// TwinCAT 3 PLC project Test_Proj
// ProgramVersion: 3.1.4026.25
// libraries:
//   Base Library, * (Beckhoff UK)
//   Eventlogger Library, * (Beckhoff UK)
//   Tc2_MC2, * (Beckhoff Automation GmbH)
//   Tc2_Standard, * (Beckhoff Automation GmbH)
//   Tc2_System, * (Beckhoff Automation GmbH)
//   Tc3_PlcTestSuite, * (Simmel)
//   [Motion Library], * (Beckhoff UK)
// project tree:
//   Manual Testing/ IntegrationTestSuite.TcPOU
//   / PlcTask.TcTTO
//   POUs/ MAIN.TcPOU
//   TestSuites/ AxisAbsTestSuite.TcPOU, AxisHaltTestSuite.TcPOU, AxisJogTestSuite.TcPOU, AxisModTestSuite.TcPOU, AxisPowerTestSuite.TcPOU, AxisRelTestSuite.TcPOU, AxisResetTestSuite.TcPOU, AxisTestSuite.TcPOU, GearOperationTestSuite.TcPOU, AxisVelocityTestSuite.TcPOU, SoEResetTestSuite.TcPOU
//   Stubs/ StubTask.TcPOU
// real-time tasks:
//   TASK PlcTask: cycle T#10ms, priority 20, ADS port 350
// motion (NC):
//   TASK NC-Task 1 SAF: cycle T#2ms, priority 4, ADS port 501
//   TASK NC-Task 1 SVB: cycle T#10ms, priority 8, ADS port 511
//   AXIS Axis 1 (id 1)
//     General: UnitName=°
//     Dynamic: Acceleration=90000, Deceleration=90000, Jerk=270000
//     Velo: RefSearch=600, RefSync=600, SlowManual=3000, FastManual=18000, Fast=60000, Maximum=60000
//     OtherSettings: AllowMotionCmdToSlave=true
//     encoder EncType=19
//       EncPara: ScaleFactorNumerator=360, ScaleFactorDenominator=1048576, MaxCount=#xffffffff
//     drive DrvType=16
//       DrvPara: MaxCount=#xffffffff, DriveControlDWord=#x00020100
//         Analog: VeloReferenz=66000, VeloScale=32, TorqueSetpointScale=10, ScaleFactorActTorque=0.1
//         TimeComp: TaskDelayCycles=1
//     controller CtrType=1
//       CtrPara: PriorControlFactor=1
//         Observer: BandWidth=20
//   AXIS Axis 2 (id 2)
//     OtherSettings: AllowMotionCmdToSlave=true
//     encoder EncType=1
//     drive DrvType=5
//       Analog: TorqueSetpointScale=10, ScaleFactorActTorque=0.1
//     controller CtrType=1
//       CtrPara: PriorControlFactor=1
//         Observer: BandWidth=20
// I/O:
//   DEVICE Device 2 (EtherCAT), AmsNetId 10.201.62.134.3.1
//     Term 1 (EK1100) [EK1100 EtherCAT Coupler (2A E-Bus)]
//       Term 2 (EL9227-5500) [EL9227-5500 Overcurrent protection 24V DC, 2Ch., max. 10A (sum), adjustable, extended functionalities]
//       Term 3 (EL1004) [EL1004 4Ch. Dig. Input 24V, 3ms]
//       Term 4 (EL2004) [EL2004 4Ch. Dig. Output 24V, 0.5A]
//       Term 5 (EL7211-0010) [EL7211-0010 1Ch. MDP742 Servo motor output stage with OCT (50V, 4.5A RMS)]
//       Term 6 (EL9011) [EL9011 End Terminal]
// variable links:
//   (this object) <-> Device 2 (EtherCAT)/Term 1 (EK1100)/Term 5 (EL7211-0010)
//     Drive/Inputs/In/nDataIn1 <-> DRV Following error actual value/Following error actual value
//     Drive/Inputs/In/nDcOutputTime <-> InfoData/DcOutputShift
//     Drive/Inputs/In/nState1 <-> DRV Statusword/Statusword
//     Drive/Inputs/In/nState2 <-> DRV Statusword/Statusword @bit 8
//     Drive/Inputs/In/nState4 @bit 1 <-> WcState/InputToggle
//     Drive/Inputs/In/nState4 <-> WcState/WcState
//     Drive/Outputs/Out/nCtrl1 <-> DRV Controlword/Controlword
//     Drive/Outputs/Out/nCtrl2 <-> DRV Controlword/Controlword @bit 8
//     Drive/Outputs/Out/nDataOut1 <-> DRV Target position/Target position
//     Enc/Inputs/In/nDataIn1 <-> FB Position/Position
//     Enc/Inputs/In/nDcInputTime <-> InfoData/DcInputShift
//     Enc/Inputs/In/nState4 @bit 1 <-> WcState/InputToggle
//     Enc/Inputs/In/nState4 <-> WcState/WcState
//   Test_Proj Instance <-> NC-Task 1 SAF/Axes/Axis 1
//     PlcTask Inputs/MAIN.Integration_TestSuite.StubAxis.NcToPlc <-> Outputs/ToPlc
//     PlcTask Outputs/MAIN.Integration_TestSuite.StubAxis.PlcToNc <-> Inputs/FromPlc
//   Test_Proj Instance <-> NC-Task 1 SAF/Axes/Axis 2
//     PlcTask Inputs/MAIN.Integration_TestSuite.gearSlave.NcToPlc <-> Outputs/ToPlc
//     PlcTask Outputs/MAIN.Integration_TestSuite.gearSlave.PlcToNc <-> Inputs/FromPlc
//   Test_Proj Instance <-> Test_Proj/Test_Proj Instance
//     PlcTask Inputs/MAIN.GearOperation_TestSuite.StubAxisRef1.NcToPlc/CoupleState <-> PlcTask Outputs/MAIN.GearOperation_TestSuite.GearAxisCoupledFeedback
//     PlcTask Inputs/MAIN.GearOperation_TestSuite.StubAxisRef1.NcToPlc/StateDWord <-> PlcTask Outputs/MAIN.GearOperation_TestSuite.GearAxisMotionFeedback
//     PlcTask Inputs/MAIN.Halt_TestSuite.StubAxis.NcToPlc/StateDWord <-> PlcTask Outputs/MAIN.Halt_TestSuite.HaltAxisStatusFeedback
//     PlcTask Outputs/MAIN.GearOperation_TestSuite.GearAxisCoupledFeedback <-> PlcTask Inputs/MAIN.GearOperation_TestSuite.StubAxisRef1.NcToPlc/CoupleState
//     PlcTask Outputs/MAIN.GearOperation_TestSuite.GearAxisMotionFeedback <-> PlcTask Inputs/MAIN.GearOperation_TestSuite.StubAxisRef1.NcToPlc/StateDWord
//     PlcTask Outputs/MAIN.Halt_TestSuite.HaltAxisStatusFeedback <-> PlcTask Inputs/MAIN.Halt_TestSuite.StubAxis.NcToPlc/StateDWord

CONFIGURATION Test_Proj
    RESOURCE PLC ON TwinCAT3
        TASK PlcTask(INTERVAL := T#10ms, PRIORITY := 20);
        PROGRAM MAIN WITH PlcTask : MAIN;
    END_RESOURCE
END_CONFIGURATION

// ---- POUs/MAIN.TcPOU
PROGRAM MAIN
VAR
	Power_TestSuite : AxisPowerTestSuite;
	Reset_TestSuite : AxisResetTestSuite;
	Halt_TestSuite : AxisHaltTestSuite;
	Axis_TestSuite : AxisTestSuite;
	AxisJog_TestSuite : AxisJogTestSuite;
	AxisVelo_TestSuite : AxisVelocityTestSuite;
	AxisAbs_TestSuite : AxisAbsTestSuite;
	AxisMod_TestSuite : AxisModTestSuite;
	AxisRel_TestSuite : AxisRelTestSuite;
	GearOperation_TestSuite : GearOperationTestSuite;
	SoEReset_TestSuite : SoEResetTestSuite;
	ReRun: BOOL;
	i : INT;
	Integration_TestSuite : IntegrationTestSuite;
END_VAR

Power_TestSuite();
Reset_TestSuite();
Halt_TestSuite();
Axis_TestSuite();
AxisJog_TestSuite();
AxisVelo_TestSuite();
AxisAbs_TestSuite();
AxisMod_TestSuite();
AxisRel_TestSuite();
GearOperation_TestSuite();
SoEReset_TestSuite();

Integration_TestSuite();

END_PROGRAM

// ---- TestSuites/AxisPowerTestSuite.TcPOU
FUNCTION_BLOCK AxisPowerTestSuite
VAR
	StubAxis : AXIS_REF;
	iStubTask : I_Task;
	TestAxisPower : EnableDisableTask := (AxisRef := StubAxis);
	ObjTestSuite : TestSuite<TestSuiteParameter.MaxTestCount>(ResultFile := JUnitResultFile) := (TestSuiteName := 'Object Test Suite');
END_VAR

DoesAxisAcceptEnable_Test();
RejectDisableWhenDisabled_Test();
RejectEnableWhenEnabled_Test();

METHOD DoesAxisAcceptEnable_Test : BOOL
VAR_INST
	Expected : BOOL := TRUE;
	Actual	 : BOOL;
END_VAR
IF ObjTestSuite.Test(__POUNAME()).ExecuteTest() THEN
	Actual := SUCCEEDED(TestAxisPower.Enable());
	TestAxisPower.Disable();
	ObjTestSuite.Test(__POUNAME()).AssertEqual(Expected, Actual);
END_IF
END_METHOD

METHOD RejectDisableWhenDisabled_Test : BOOL
VAR_INST
	Expected : BOOL := TRUE;
	Actual	 : BOOL;
END_VAR
IF ObjTestSuite.Test(__POUNAME()).ExecuteTest() THEN
	Actual := FAILED(TestAxisPower.Disable());
	ObjTestSuite.Test(__POUNAME()).AssertEqual(Expected, Actual);
END_IF
END_METHOD

METHOD RejectEnableWhenEnabled_Test : BOOL
VAR_INST
	Expected : BOOL := TRUE;
	Actual	 : BOOL;
END_VAR
IF ObjTestSuite.Test(__POUNAME()).ExecuteTest() THEN
	TestAxisPower.Enable();
	Actual := FAILED(TestAxisPower.Enable());
	TestAxisPower.Abort();
	ObjTestSuite.Test(__POUNAME()).AssertEqual(Expected, Actual);
END_IF
END_METHOD

END_FUNCTION_BLOCK

// ---- TestSuites/AxisResetTestSuite.TcPOU
FUNCTION_BLOCK AxisResetTestSuite 
VAR
	StubAxis : AXIS_REF;
	iStubTask : I_Task;
	TestAxisReset : CoEResetTask := (AxisRef := StubAxis);
	ObjTestSuite : TestSuite<TestSuiteParameter.MaxTestCount>(ResultFile := JUnitResultFile) := (TestSuiteName := 'Object Test Suite');
END_VAR

DoesAcceptExecute_Test();
DoesTaskAbortClearBusy_Test();
DoesTaskAccept_Test();
RejectResetWhileResetting_Test();

METHOD DoesAcceptExecute_Test : BOOL
VAR_INST
	Expected : HRESULT;
	Actual	 : HRESULT;
END_VAR
IF ObjTestSuite.Test(__POUNAME()).ExecuteTest() THEN
	Expected := s_OK;
	Actual := TestAxisReset.Reset();
	TestAxisReset.Abort();
	ObjTestSuite.Test(__POUNAME()).AssertEqual(Expected, Actual);
END_IF
END_METHOD

METHOD DoesTaskAbortClearBusy_Test
VAR_INST
	Expected : BOOL := FALSE;
	Actual	 : BOOL;
END_VAR
IF ObjTestSuite.Test(__POUNAME()).ExecuteTest() THEN
	TestAxisReset.Reset();
	TestAxisReset.Abort();
	Actual := TestAxisReset.Busy;
	ObjTestSuite.Test(__POUNAME()).AssertEqual(Expected, Actual);
END_IF
END_METHOD

METHOD DoesTaskAccept_Test
VAR_INST
	Expected : BOOL := TRUE;
	Actual	 : bool;
END_VAR
IF ObjTestSuite.Test(__POUNAME()).ExecuteTest() THEN
	Actual := SUCCEEDED(TestAxisReset.Reset());
	TestAxisReset.Abort();
	ObjTestSuite.Test(__POUNAME()).AssertEqual(Expected, Actual);
END_IF
END_METHOD

METHOD RejectResetWhileResetting_Test : BOOL
VAR_INST
	Expected : BOOL := TRUE;
	Actual	 : BOOL;
END_VAR
IF ObjTestSuite.Test(__POUNAME()).ExecuteTest() THEN
	TestAxisReset.Reset();
	Actual := FAILED(TestAxisReset.Reset());
	ObjTestSuite.Test(__POUNAME()).AssertEqual(Expected, Actual);
END_IF
END_METHOD

END_FUNCTION_BLOCK

// ---- TestSuites/AxisHaltTestSuite.TcPOU
FUNCTION_BLOCK AxisHaltTestSuite
VAR
	StubAxis : AXIS_REF;
	iStubTask : I_Task;
	TestAxisHalt : HaltTask := (AxisRef := StubAxis);
	HaltAxisStatusFeedback AT%Q* : DWORD;
	Cycle : INT;
	ObjTestSuite : TestSuite<TestSuiteParameter.MaxTestCount>(ResultFile := JUnitResultFile) := (TestSuiteName := 'Object Test Suite');
END_VAR

CASE Cycle OF
	0:
		DoesTaskAbortClearBusy_Test();
		DoesTaskAcceptDeceleration_Test();
		DoesTaskAcceptJerk_Test();
		DoesTaskRejectHaltWhenHalting_Test();
		DoesTaskRejectHaltWhenStationary();
		DoesTaskRejectNegativeDecel_Test();
		DoesTaskRejectNegativeJerk_Test();
		HaltAxisStatusFeedback := 512;
		IF StubAxis.Status.Moving THEN
			Cycle := 1;
		END_IF
		
	1:
		DoesTaskAcceptHaltSettingBusy();
		HaltAxisStatusFeedback := 0;
		Cycle := 0;
END_CASE

StubAxis.ReadStatus();

METHOD DoesTaskAbortClearBusy_Test
VAR_INST
	Expected : BOOL := False;
	Actual	 : BOOL;
END_VAR
IF ObjTestSuite.Test(__POUNAME()).ExecuteTest() THEN
	TestAxisHalt.Execute();
	TestAxisHalt.Abort();
	Actual := TestAxisHalt.Busy;
	ObjTestSuite.Test(__POUNAME()).AssertEqual(Expected, Actual);
END_IF
END_METHOD

METHOD DoesTaskAcceptDeceleration_Test
VAR_INST
	Expected : BOOL := TRUE;
	Actual	 : BOOL;
END_VAR
IF ObjTestSuite.Test(__POUNAME()).ExecuteTest() THEN
	TestAxisHalt.Deceleration := 1.0;
	Actual := TestAxisHalt.Deceleration = 1.0;
	ObjTestSuite.Test(__POUNAME()).AssertEqual(Expected, Actual);
	TestAxisHalt.Deceleration := 0.0;
	TestAxisHalt.Abort();
END_IF
END_METHOD

METHOD DoesTaskAcceptHaltSettingBusy
VAR_INST
	Expected : BOOL := TRUE;
	Actual	 : BOOL;
END_VAR
IF ObjTestSuite.Test(__POUNAME()).ExecuteTest() THEN
	TestAxisHalt.Execute();
	Actual := TestAxisHalt.Busy;
	ObjTestSuite.Test(__POUNAME()).AssertEqual(Expected, Actual);
	TestAxisHalt.Abort();
	HaltAxisStatusFeedback := 0;
END_IF
END_METHOD

METHOD DoesTaskAcceptJerk_Test
VAR_INST
	Expected : BOOL := TRUE;
	Actual	 : BOOL;
END_VAR
IF ObjTestSuite.Test(__POUNAME()).ExecuteTest() THEN
	TestAxisHalt.Jerk := 1.0;
	Actual := TestAxisHalt.Jerk = 1.0;
	ObjTestSuite.Test(__POUNAME()).AssertEqual(Expected, Actual);
	TestAxisHalt.Jerk := 0.0;
	TestAxisHalt.Abort();
END_IF
END_METHOD

METHOD DoesTaskRejectHaltWhenHalting_Test : BOOL
VAR_INST
	Expected : HRESULT;
	Actual	 : HRESULT;
END_VAR
IF ObjTestSuite.Test(__POUNAME()).ExecuteTest() THEN
	Expected := S_FALSE;
	TestAxisHalt.Execute();
	Actual := TestAxisHalt.Execute();
	ObjTestSuite.Test(__POUNAME()).AssertEqual(Expected, Actual);
	TestAxisHalt.Abort();
END_IF
END_METHOD

METHOD DoesTaskRejectHaltWhenStationary : BOOL
VAR_INST
	Expected : HRESULT;
	Actual	 : HRESULT;
END_VAR
IF ObjTestSuite.Test(__POUNAME()).ExecuteTest() THEN
	Expected := S_FALSE;
	Actual := TestAxisHalt.Execute();
	ObjTestSuite.Test(__POUNAME()).AssertEqual(Expected, Actual);
	TestAxisHalt.Abort();
END_IF
END_METHOD

METHOD DoesTaskRejectNegativeDecel_Test
VAR_INST
	Expected : BOOL := TRUE;
	Actual	 : BOOL;
END_VAR
IF ObjTestSuite.Test(__POUNAME()).ExecuteTest() THEN
	TestAxisHalt.Deceleration := -1.0;
	Actual := TestAxisHalt.Deceleration = 0.0;
	ObjTestSuite.Test(__POUNAME()).AssertEqual(Expected, Actual);
	TestAxisHalt.Abort();
END_IF
END_METHOD

METHOD DoesTaskRejectNegativeJerk_Test
VAR_INST
	Expected : BOOL := TRUE;
	Actual	 : BOOL;
END_VAR
IF ObjTestSuite.Test(__POUNAME()).ExecuteTest() THEN
	TestAxisHalt.Jerk := -1.0;
	Actual := TestAxisHalt.jerk = 0.0;
	ObjTestSuite.Test(__POUNAME()).AssertEqual(Expected, Actual);
	TestAxisHalt.Abort();
END_IF
END_METHOD

END_FUNCTION_BLOCK

// ---- TestSuites/AxisTestSuite.TcPOU
FUNCTION_BLOCK AxisTestSuite
VAR
	StubAxis : AXIS_REF;
	TestAxis : Axis_Base(StubAxis);
 	DummyLogger : Message_Null;
	ObjTestSuite : TestSuite<TestSuiteParameter.MaxTestCount>(ResultFile := JUnitResultFile) := (TestSuiteName := 'Object Test Suite');
END_VAR

AxisPassesEnableRequest_Test();

METHOD AxisPassesEnableRequest_Test
VAR_INST
	Expected : BOOL := TRUE;
	Actual	 : BOOL;
END_VAR
IF ObjTestSuite.Test(__POUNAME()).ExecuteTest() THEN
	Actual := SUCCEEDED(TestAxis.EnableAxis(FALSE,FALSE));
	ObjTestSuite.Test(__POUNAME()).AssertEqual(Expected, Actual);
END_IF
END_METHOD

END_FUNCTION_BLOCK

// ---- TestSuites/AxisJogTestSuite.TcPOU
FUNCTION_BLOCK AxisJogTestSuite
VAR
	StubAxis : AXIS_REF;
	iStubTask : I_Task;
	TestAxisJog : JogTask := (AxisRef := stubaxis);
	ObjTestSuite : TestSuite<TestSuiteParameter.MaxTestCount>(ResultFile := JUnitResultFile) := (TestSuiteName := 'Object Test Suite');
END_VAR

DoesTaskAcceptAcceleration_Test();
DoesTaskAcceptDeceleration_Test();
DoesTaskAcceptJerk_Test();
DoesTaskAcceptsInch_Test();
DoesTaskRejectNegativeAccell_Test();
DoesTaskRejectNegativeDecel_Test();
DoesTaskRejectNegativeJerk_Test();
DoesTaskRejectZeroDistanceInch_Test();

METHOD DoesTaskAcceptAcceleration_Test
VAR_INST
	Expected : BOOL := TRUE;
	Actual	 : BOOL;
END_VAR
IF ObjTestSuite.Test(__POUNAME()).ExecuteTest() THEN
	TestAxisJog.Acceleration := 1.0;
	Actual := TestAxisJog.Acceleration = 1.0;
	ObjTestSuite.Test(__POUNAME()).AssertEqual(Expected, Actual);
	TestAxisJog.Acceleration := 0.0;
	TestAxisJog.Abort();
END_IF
END_METHOD

METHOD DoesTaskAcceptDeceleration_Test
VAR_INST
	Expected : BOOL := TRUE;
	Actual	 : BOOL;
END_VAR
IF ObjTestSuite.Test(__POUNAME()).ExecuteTest() THEN
	TestAxisJog.Deceleration := 1.0;
	Actual := TestAxisJog.Deceleration = 1.0;
	ObjTestSuite.Test(__POUNAME()).AssertEqual(Expected, Actual);
	TestAxisJog.Deceleration := 0.0;
	TestAxisJog.Abort();
END_IF
END_METHOD

METHOD DoesTaskAcceptJerk_Test
VAR_INST
	Expected : BOOL := TRUE;
	Actual	 : BOOL;
END_VAR
IF ObjTestSuite.Test(__POUNAME()).ExecuteTest() THEN
	TestAxisJog.Jerk := 1.0;
	Actual := TestAxisJog.Jerk = 1.0;
	ObjTestSuite.Test(__POUNAME()).AssertEqual(Expected, Actual);
	TestAxisJog.Jerk := 0.0;
	TestAxisJog.Abort();
END_IF
END_METHOD

METHOD DoesTaskAcceptsInch_Test
VAR_INST
	Expected : BOOL := TRUE;
	Actual	 : BOOL;
END_VAR
IF ObjTestSuite.Test(__POUNAME()).ExecuteTest() THEN
	Actual := SUCCEEDED(TestAxisJog.Inch(10.0,TRUE));
	ObjTestSuite.Test(__POUNAME()).AssertEqual(Expected, Actual);
	TestAxisJog.Abort();
END_IF
END_METHOD

METHOD DoesTaskRejectNegativeAccell_Test
VAR_INST
	Expected : BOOL := TRUE;
	Actual	 : BOOL;
END_VAR
IF ObjTestSuite.Test(__POUNAME()).ExecuteTest() THEN
	TestAxisJog.Acceleration := -1.0;
	Actual := TestAxisJog.Acceleration = 0.0;
	ObjTestSuite.Test(__POUNAME()).AssertEqual(Expected, Actual);
	TestAxisJog.Abort();
END_IF
END_METHOD

METHOD DoesTaskRejectNegativeDecel_Test
VAR_INST
	Expected : BOOL := TRUE;
	Actual	 : BOOL;
END_VAR
IF ObjTestSuite.Test(__POUNAME()).ExecuteTest() THEN
	TestAxisJog.Deceleration := -1.0;
	Actual := TestAxisJog.Deceleration = 0.0;
	ObjTestSuite.Test(__POUNAME()).AssertEqual(Expected, Actual);
	TestAxisJog.Abort();
END_IF
END_METHOD

METHOD DoesTaskRejectNegativeJerk_Test
VAR_INST
	Expected : BOOL := TRUE;
	Actual	 : BOOL;
END_VAR
IF ObjTestSuite.Test(__POUNAME()).ExecuteTest() THEN
	TestAxisJog.Jerk := -1.0;
	Actual := TestAxisJog.jerk = 0.0;
	ObjTestSuite.Test(__POUNAME()).AssertEqual(Expected, Actual);
	TestAxisJog.Abort();
END_IF
END_METHOD

METHOD DoesTaskRejectZeroDistanceInch_Test
VAR_INST
	Expected : BOOL := TRUE;
	Actual	 : BOOL;
END_VAR
IF ObjTestSuite.Test(__POUNAME()).ExecuteTest() THEN
	Actual := FAILED(TestAxisJog.Inch(-10.0,TRUE));
	ObjTestSuite.Test(__POUNAME()).AssertEqual(Expected, Actual);
	TestAxisJog.Abort();
END_IF
END_METHOD

END_FUNCTION_BLOCK

// ---- TestSuites/AxisVelocityTestSuite.TcPOU
FUNCTION_BLOCK AxisVelocityTestSuite 
VAR
	StubAxis : AXIS_REF;
	iStubTask : I_Task;
	TestAxisVelo : MoveVeloTask := (AxisRef := StubAxis);
	ObjTestSuite : TestSuite<TestSuiteParameter.MaxTestCount>(ResultFile := JUnitResultFile) := (TestSuiteName := 'Object Test Suite');
END_VAR

DoesTaskAcceptAcceleration_Test();
DoesTaskAcceptDeceleration_Test();
DoesTaskAcceptJerk_Test();
DoesTaskRejectAZeroVelocity_Test();
DoesTaskRejectNegativeAccell_Test();
DoesTaskRejectNegativeDecel_Test();
DoesTaskRejectNegativeJerk_Test();
DoesTaskRejectNegativeVelocity_Test();

METHOD DoesTaskAcceptAcceleration_Test
VAR_INST
	Expected : BOOL := TRUE;
	Actual	 : BOOL;
END_VAR
IF ObjTestSuite.Test(__POUNAME()).ExecuteTest() THEN
	TestAxisVelo.Acceleration := 1.0;
	Actual := TestAxisVelo.Acceleration = 1.0;
	ObjTestSuite.Test(__POUNAME()).AssertEqual(Expected, Actual);
	TestAxisVelo.Acceleration := 0.0;
	TestAxisVelo.Abort();
END_IF
END_METHOD

METHOD DoesTaskAcceptDeceleration_Test
VAR_INST
	Expected : BOOL := TRUE;
	Actual	 : BOOL;
END_VAR
IF ObjTestSuite.Test(__POUNAME()).ExecuteTest() THEN
	TestAxisVelo.Deceleration := 1.0;
	Actual := TestAxisVelo.Deceleration = 1.0;
	ObjTestSuite.Test(__POUNAME()).AssertEqual(Expected, Actual);
	TestAxisVelo.Deceleration := 0.0;
	TestAxisVelo.Abort();
END_IF
END_METHOD

METHOD DoesTaskAcceptJerk_Test
VAR_INST
	Expected : BOOL := TRUE;
	Actual	 : BOOL;
END_VAR
IF ObjTestSuite.Test(__POUNAME()).ExecuteTest() THEN
	TestAxisVelo.Jerk := 1.0;
	Actual := TestAxisVelo.Jerk = 1.0;
	ObjTestSuite.Test(__POUNAME()).AssertEqual(Expected, Actual);
	TestAxisVelo.Jerk := 0.0;
	TestAxisVelo.Abort();
END_IF
END_METHOD

METHOD DoesTaskRejectAZeroVelocity_Test
VAR_INST
	Expected : BOOL := TRUE;
	Actual	 : BOOL;
END_VAR
IF ObjTestSuite.Test(__POUNAME()).ExecuteTest() THEN
	iStubTask := 0;
	Actual := FAILED(TestAxisVelo.MoveAtVelocity(mc_direction.MC_Positive_Direction, 0.0));
	ObjTestSuite.Test(__POUNAME()).AssertEqual(Expected, Actual);
	TestAxisVelo.Abort();
END_IF
END_METHOD

METHOD DoesTaskRejectNegativeAccell_Test
VAR_INST
	Expected : BOOL := TRUE;
	Actual	 : BOOL;
END_VAR
IF ObjTestSuite.Test(__POUNAME()).ExecuteTest() THEN
	TestAxisVelo.Acceleration := -1.0;
	Actual := TestAxisVelo.Acceleration = 0.0;
	ObjTestSuite.Test(__POUNAME()).AssertEqual(Expected, Actual);
	TestAxisVelo.Abort();
END_IF
END_METHOD

METHOD DoesTaskRejectNegativeDecel_Test
VAR_INST
	Expected : BOOL := TRUE;
	Actual	 : BOOL;
END_VAR
IF ObjTestSuite.Test(__POUNAME()).ExecuteTest() THEN
	TestAxisVelo.Deceleration := -1.0;
	Actual := TestAxisVelo.Deceleration = 0.0;
	ObjTestSuite.Test(__POUNAME()).AssertEqual(Expected, Actual);
	TestAxisVelo.Abort();
END_IF
END_METHOD

METHOD DoesTaskRejectNegativeJerk_Test
VAR_INST
	Expected : BOOL := TRUE;
	Actual	 : BOOL;
END_VAR
IF ObjTestSuite.Test(__POUNAME()).ExecuteTest() THEN
	TestAxisVelo.Jerk := -1.0;
	Actual := TestAxisVelo.jerk = 0.0;
	ObjTestSuite.Test(__POUNAME()).AssertEqual(Expected, Actual);
	TestAxisVelo.Abort();
END_IF
END_METHOD

METHOD DoesTaskRejectNegativeVelocity_Test
VAR_INST
	Expected : BOOL := TRUE;
	Actual	 : BOOL;
END_VAR
IF ObjTestSuite.Test(__POUNAME()).ExecuteTest() THEN
	iStubTask := 0;
	Actual := FAILED(TestAxisVelo.MoveAtVelocity(mc_direction.MC_Positive_Direction, -70.0));
	ObjTestSuite.Test(__POUNAME()).AssertEqual(Expected, Actual);
	TestAxisVelo.Abort();
END_IF
END_METHOD

END_FUNCTION_BLOCK

// ---- TestSuites/AxisAbsTestSuite.TcPOU
FUNCTION_BLOCK AxisAbsTestSuite
VAR
	StubAxis : AXIS_REF;
	iStubTask : I_Task;
	TestAxisAbs : MoveAbsTask := (AxisRef := stubaxis);
	TestObjRunner : ObjectRunner<99>;
	ObjTestSuite : TestSuite<TestSuiteParameter.MaxTestCount>(ResultFile := JUnitResultFile) := (TestSuiteName := 'Object Test Suite');
END_VAR

CheckCorrectRegistration_Test();
TaskAcceptValidCommand_Test();
TaskRejectsZeroVeloCommand_Test();

METHOD CheckCorrectRegistration_Test : BOOL
VAR_INST
	Expected : BOOL := TRUE;
	Actual	 : bool;
END_VAR
IF ObjTestSuite.Test(__POUNAME()).ExecuteTest() THEN
	TestAxisAbs.RegisterWithParent(TestObjRunner);
	Actual := TestObjRunner.CyclicModuleCount = TestObjRunner.AbortableModuleCount AND
				TestObjRunner.CyclicModuleCount = TestObjRunner.TaskModuleCount;
	ObjTestSuite.Test(__POUNAME()).AssertEqual(Expected, Actual);
END_IF
END_METHOD

METHOD TaskAcceptValidCommand_Test : BOOL
VAR_INST
	Expected : BOOL := TRUE;
	Actual	 : BOOL;
END_VAR
IF ObjTestSuite.Test(__POUNAME()).ExecuteTest() THEN
	Actual := SUCCEEDED(TestAxisAbs.MoveTo(100.0, 300.0));
	TestAxisAbs.Abort();
	ObjTestSuite.Test(__POUNAME()).AssertEqual(Expected, Actual);
END_IF
END_METHOD

METHOD TaskRejectsZeroVeloCommand_Test : BOOL
VAR_INST
	Expected : BOOL := TRUE;
	Actual	 : BOOL;
END_VAR
IF ObjTestSuite.Test(__POUNAME()).ExecuteTest() THEN
	Actual := FAILED(TestAxisAbs.MoveTo(100.0, 0.0));
	TestAxisAbs.Abort();
	ObjTestSuite.Test(__POUNAME()).AssertEqual(Expected, Actual);
END_IF
END_METHOD

END_FUNCTION_BLOCK

// ---- TestSuites/AxisModTestSuite.TcPOU
FUNCTION_BLOCK AxisModTestSuite
VAR
	StubAxis : AXIS_REF;
	iStubTask : I_Task;
	TestAxisMod : MoveModTask := (AxisRef := stubaxis);
	TestObjRunner : ObjectRunner<99>;
	ObjTestSuite : TestSuite<TestSuiteParameter.MaxTestCount>(ResultFile := JUnitResultFile) := (TestSuiteName := 'Object Test Suite');
END_VAR

CheckCorrectRegistration_Test();
TaskAcceptValidCommand_Test();
TaskRejectsZeroVeloCommand_Test();

METHOD CheckCorrectRegistration_Test : BOOL
VAR_INST
	Expected : BOOL := TRUE;
	Actual	 : bool;
END_VAR
IF ObjTestSuite.Test(__POUNAME()).ExecuteTest() THEN
	TestAxisMod.RegisterWithParent(TestObjRunner);
	Actual := TestObjRunner.CyclicModuleCount = TestObjRunner.AbortableModuleCount AND
				TestObjRunner.CyclicModuleCount = TestObjRunner.TaskModuleCount;
	ObjTestSuite.Test(__POUNAME()).AssertEqual(Expected, Actual);
END_IF
END_METHOD

METHOD TaskAcceptValidCommand_Test : BOOL
VAR_INST
	Expected : BOOL := TRUE;
	Actual	 : BOOL;
END_VAR
IF ObjTestSuite.Test(__POUNAME()).ExecuteTest() THEN
	Actual := SUCCEEDED(TestAxisMod.MoveTo(100.0, 300.0));
	TestAxisMod.Abort();
	ObjTestSuite.Test(__POUNAME()).AssertEqual(Expected, Actual);
END_IF
END_METHOD

METHOD TaskRejectsZeroVeloCommand_Test : BOOL
VAR_INST
	Expected : BOOL := TRUE;
	Actual	 : BOOL;
END_VAR
IF ObjTestSuite.Test(__POUNAME()).ExecuteTest() THEN
	Actual := FAILED(TestAxisMod.MoveTo(100.0, 0.0));
	TestAxisMod.Abort();
	ObjTestSuite.Test(__POUNAME()).AssertEqual(Expected, Actual);
END_IF
END_METHOD

END_FUNCTION_BLOCK

// ---- TestSuites/AxisRelTestSuite.TcPOU
FUNCTION_BLOCK AxisRelTestSuite 
VAR
	StubAxis : AXIS_REF;
	iStubTask : I_Task;
	TestAxisRel : MoveRelTask := (AxisRef := stubaxis);
	TestObjRunner : ObjectRunner<99>;
	ObjTestSuite : TestSuite<TestSuiteParameter.MaxTestCount>(ResultFile := JUnitResultFile) := (TestSuiteName := 'Object Test Suite');
END_VAR

CheckCorrectRegistration_Test();
TaskAcceptValidCommand_Test();
TaskRejectsZeroVeloCommand_Test();

METHOD CheckCorrectRegistration_Test : BOOL
VAR_INST
	Expected : BOOL := TRUE;
	Actual	 : bool;
END_VAR
IF ObjTestSuite.Test(__POUNAME()).ExecuteTest() THEN
	TestAxisRel.RegisterWithParent(TestObjRunner);
	Actual := TestObjRunner.CyclicModuleCount = TestObjRunner.AbortableModuleCount AND
				TestObjRunner.CyclicModuleCount = TestObjRunner.TaskModuleCount;
	ObjTestSuite.Test(__POUNAME()).AssertEqual(Expected, Actual);
END_IF
END_METHOD

METHOD TaskAcceptValidCommand_Test : BOOL
VAR_INST
	Expected : BOOL := TRUE;
	Actual	 : bool;
END_VAR
IF ObjTestSuite.Test(__POUNAME()).ExecuteTest() THEN
	Actual := SUCCEEDED(TestAxisRel.MoveBy(100.0, 300.0));
	TestAxisRel.Abort();
	ObjTestSuite.Test(__POUNAME()).AssertEqual(Expected, Actual);
END_IF
END_METHOD

METHOD TaskRejectsZeroVeloCommand_Test : BOOL
VAR_INST
	Expected : BOOL := TRUE;
	Actual	 : bool;
END_VAR
IF ObjTestSuite.Test(__POUNAME()).ExecuteTest() THEN
	Actual := FAILED(TestAxisRel.MoveBy(100.0, 0.0));
	TestAxisRel.Abort();
	ObjTestSuite.Test(__POUNAME()).AssertEqual(Expected, Actual);
END_IF
END_METHOD

END_FUNCTION_BLOCK

// ---- TestSuites/GearOperationTestSuite.TcPOU
FUNCTION_BLOCK GearOperationTestSuite
VAR
	StubAxisRef1 : AXIS_REF;
	StubAxisRef2 : AXIS_REF;
	StubSlave : Axis_Base(StubAxisRef1);
	StubMaster : Axis_Base(StubAxisRef2);
	GearAxisCoupledFeedback AT%Q* : UDINT := 0;
	GearAxisMotionFeedback AT%Q* : DWORD;
	TestState : INT := 0;
	ObjTestSuite : TestSuite<TestSuiteParameter.MaxTestCount>(ResultFile := JUnitResultFile) := (TestSuiteName := 'Object Test Suite');
END_VAR

CASE TestState OF
	0:
		OperationRejectsCommandsWithNoAxes_Test();
		OperationRejectsDuplicateGearCommand_Test();
		OperationRejectsDupicateUnGearCommand_Test();
		OperationRejectsUnGearWhenNotCoupled_Test();
		GearAxisCoupledFeedback := 3;
		IF StubAxisRef1.Status.Coupled THEN
			TestState := 1;	
		END_IF
		
	1:
		OperationRejectsGearWhenCoupled_Test();
		GearAxisMotionFeedback := 512;
		GearAxisCoupledFeedback := 0;
		IF StubAxisRef1.Status.Moving THEN
			TestState := 2;	
		END_IF	
	2:
		OperationsRejectsGearWhenNotStationary_Test();
		TestState := 0;
		GearAxisMotionFeedback := 0;
END_CASE


StubAxisRef1.ReadStatus();
StubAxisRef2.ReadStatus();

METHOD OperationRejectsCommandsWithNoAxes_Test : BOOL
VAR_INST
	TestGearOperation : GearAxes;
	Expected : BOOL := TRUE;
	Actual	 : BOOL;
END_VAR
IF ObjTestSuite.Test(__POUNAME()).ExecuteTest() THEN
	Actual := FAILED(TestGearOperation.GearIn());
	TestGearOperation.Abort();
	ObjTestSuite.Test(__POUNAME()).AssertEqual(Expected, Actual);
END_IF
END_METHOD

METHOD OperationRejectsDupicateUnGearCommand_Test : BOOL
VAR_INST
	TestGearOperation : GearAxes := (Slave := StubSlave, Master := StubMaster);
	Expected : BOOL := TRUE;
	Actual	 : BOOL;
END_VAR
IF ObjTestSuite.Test(__POUNAME()).ExecuteTest() THEN
	TestGearOperation.GearOut();
	Actual := FAILED(TestGearOperation.GearOut());
	TestGearOperation.Abort();
	ObjTestSuite.Test(__POUNAME()).AssertEqual(Expected, Actual);
END_IF
END_METHOD

METHOD OperationRejectsDuplicateGearCommand_Test : BOOL
VAR_INST
	TestGearOperation : GearAxes:= (Slave := StubSlave, Master := StubMaster);
	Expected : BOOL := TRUE;
	Actual	 : BOOL;
END_VAR
IF ObjTestSuite.Test(__POUNAME()).ExecuteTest() THEN
	TestGearOperation.GearIn();
	Actual := FAILED(TestGearOperation.GearIn());
	TestGearOperation.Abort();
	ObjTestSuite.Test(__POUNAME()).AssertEqual(Expected, Actual);
END_IF
END_METHOD

METHOD OperationRejectsGearWhenCoupled_Test : BOOL
VAR_INST
	TestGearOperation : GearAxes:= (Slave := StubSlave, Master := StubMaster);
	Expected : BOOL := TRUE;
	Actual	 : BOOL;
END_VAR
IF ObjTestSuite.Test(__POUNAME()).ExecuteTest() THEN
	Actual := FAILED(TestGearOperation.GearIn());
	TestGearOperation.Abort();
	ObjTestSuite.Test(__POUNAME()).AssertEqual(Expected, Actual);
END_IF
END_METHOD

METHOD OperationRejectsUnGearWhenNotCoupled_Test : BOOL
VAR_INST
	TestGearOperation : GearAxes:= (Slave := StubSlave, Master := StubMaster);
	Expected : BOOL := TRUE;
	Actual	 : BOOL;
END_VAR
IF ObjTestSuite.Test(__POUNAME()).ExecuteTest() THEN
	Actual := FAILED(TestGearOperation.GearOut());
	TestGearOperation.Abort();
	ObjTestSuite.Test(__POUNAME()).AssertEqual(Expected, Actual);
END_IF
END_METHOD

METHOD OperationsRejectsGearWhenNotStationary_Test : BOOL
VAR_INST
	TestGearOperation : GearAxes:= (Slave := StubSlave, Master := StubMaster);
	Expected : BOOL := TRUE;
	Actual	 : bool;
END_VAR
IF ObjTestSuite.Test(__POUNAME()).ExecuteTest() THEN
	Actual := FAILED(TestGearOperation.GearIn());
	TestGearOperation.Abort();
	ObjTestSuite.Test(__POUNAME()).AssertEqual(Expected, Actual);
END_IF
END_METHOD

END_FUNCTION_BLOCK

// ---- TestSuites/SoEResetTestSuite.TcPOU
FUNCTION_BLOCK SoEResetTestSuite
VAR
	StubAxis : AXIS_REF;
	iStubTask : I_Task;
	Soe_Reset : SoEResetTask;
	TestObjRunner : ObjectRunner<99>;
	ObjTestSuite : TestSuite<TestSuiteParameter.MaxTestCount>(ResultFile := JUnitResultFile) := (TestSuiteName := 'Object Test Suite');
END_VAR

TaskRejectsCycleCallWithoutAxisRef_Test();
TaskAcceptsResetCommand_Test();
TaskRejectsDuplicateResetCommand_Test();
CheckCorrectRegistration_Test();

METHOD CheckCorrectRegistration_Test : BOOL
VAR_INST
	Expected : BOOL := TRUE;
	Actual	 : BOOL;
END_VAR
IF ObjTestSuite.Test(__POUNAME()).ExecuteTest() THEN
	Soe_Reset.RegisterWithParent(TestObjRunner);
	Actual := TestObjRunner.CyclicModuleCount = TestObjRunner.AbortableModuleCount AND
				TestObjRunner.CyclicModuleCount = TestObjRunner.TaskModuleCount AND
				TestObjRunner.CyclicModuleCount = TestObjRunner.ResettableModuleCount;
	ObjTestSuite.Test(__POUNAME()).AssertEqual(Expected, Actual);
END_IF
END_METHOD

METHOD TaskAcceptsResetCommand_Test : BOOL
VAR_INST
	Expected : BOOL := TRUE;
	Actual	 : BOOL;
END_VAR
IF ObjTestSuite.Test(__POUNAME()).ExecuteTest() THEN
	Actual := SUCCEEDED(Soe_Reset.Reset());
	Soe_Reset.Abort();
	ObjTestSuite.Test(__POUNAME()).AssertEqual(Expected, Actual);
END_IF
END_METHOD

METHOD TaskRejectsCycleCallWithoutAxisRef_Test
VAR_INST
	Expected : BOOL := TRUE;
	Actual	 : BOOL;
END_VAR
IF ObjTestSuite.Test(__POUNAME()).ExecuteTest() THEN
	Actual := FAILED(Soe_Reset.Cycle());
	Soe_Reset.AxisRef REF= StubAxis;
	ObjTestSuite.Test(__POUNAME()).AssertEqual(Expected, Actual);
END_IF
END_METHOD

METHOD TaskRejectsDuplicateResetCommand_Test : BOOL
VAR_INST
	Expected : BOOL := TRUE;
	Actual	 : BOOL;
END_VAR
IF ObjTestSuite.Test(__POUNAME()).ExecuteTest() THEN
	Soe_Reset.Reset();
	Actual := FAILED(Soe_Reset.Reset());
	Soe_Reset.Abort();
	ObjTestSuite.Test(__POUNAME()).AssertEqual(Expected, Actual);
END_IF
END_METHOD

END_FUNCTION_BLOCK

// ---- Manual Testing/IntegrationTestSuite.TcPOU
FUNCTION_BLOCK IntegrationTestSuite
VAR
	StubAxis : AXIS_REF;
	gearSlave : AXIS_REF;
	TestAxis : Axis_Base(StubAxis);
	gearTestAxis : Axis_Base(gearSlave);
	iAxisBase : I_AxisBase := TestAxis;
	iJog : I_Jog := TestAxis;
	iAxisStatus : I_Status := TestAxis;
	iPosition : I_Position := TestAxis;
	iVelo : I_Velocity := TestAxis;
	gearOperation : GearAxes := (Master := TestAxis, Slave := gearTestAxis);
	Enable: BOOL;
	MOVETO: BOOL;
	MOVETWO: BOOL;
	MOVEREL : BOOL;
	DISABLE: BOOL;
	SETBUFFER: BOOL;
	CONVEYOR: BOOL;
	JOGSLOW: BOOL;
	JOGFAST: BOOL;
	HALT: BOOL;
	MODULO : BOOL;
	VelocityDemand : LREAL := 100.0;
	Pos_Dist : LREAL := 10.0;
	Mod_Pos : LREAL := 230.0;
	GEAR: BOOL;
	checkflag : BOOL;
	istartCounter: INT;
	ioperatCounter : INT;
	stationaryTest1: BOOL;
	stationaryTest2: BOOL;
END_VAR

IF Enable THEN
	IF succeeded(iAxisBase.EnableAxis(FALSE, FALSE)) AND SUCCEEDED(gearTestAxis.EnableAxis(FALSE,FALSE)) THEN
		Enable := FALSE;
	END_IF
END_IF
 IF checkflag THEN
	 istartCounter := istartCounter + 1;
 END_IF

IF iAxisBase.Operating THEN
	checkflag := FALSE;
	ioperatCounter := ioperatCounter + 1;
END_IF

IF MOVETO THEN
	IF SUCCEEDED(iPosition.MoveToPosition(1000.0,100.0)) THEN
		checkflag := TRUE;
		MOVETO := FALSE;
	END_IF
END_IF

IF SETBUFFER THEN
	SETBUFFER := FALSE;
	TestAxis.BufferMode := MC_BufferMode.MC_BlendingLow;
	
END_IF

IF MOVETWO THEN
	IF SUCCEEDED(iPosition.MoveToPosition(1200.0,VelocityDemand)) THEN
		MOVETWO := FALSE;
	END_IF
END_IF

IF MOVEREL THEN
	IF succeeded(iPosition.MoveByDistance(Pos_Dist,VelocityDemand)) THEN
		MOVEREL := FALSE;
	END_IF
END_IF

IF MODULO THEN
	IF SUCCEEDED(iPosition.MoveToModuloPosition(Mod_Pos,VelocityDemand)) THEN
		MODULO := FALSE;
	END_IF
END_IF

IF HALT THEN
	IF SUCCEEDED(iAxisBase.HaltAxis()) THEN
		HALT := FALSE;
	END_IF
END_IF

IF DISABLE THEN
	IF SUCCEEDED(iAxisBase.DisableAxis()) AND SUCCEEDED(gearTestAxis.DisableAxis()) THEN
		DISABLE := FALSE;
	END_IF
END_IF

IF GEAR THEN
	IF SUCCEEDED(gearOperation.GearIn()) THEN
		GEAR := FALSE;
	END_IF
END_IF

IF CONVEYOR THEN
	IF SUCCEEDED(iVelo.MoveAtVelocity(MC_Direction.MC_Positive_Direction, VelocityDemand)) THEN
		CONVEYOR := FALSE;
	END_IF
END_IF

IF JOGSLOW THEN
	iJog.JogSlow(FALSE);
END_IF

IF JOGFAST THEN
	iJog.JogFast(TRUE);
END_IF

stationaryTest1 := TestAxis.IsStationary;
stationaryTest2 := gearTestAxis.IsStationary;

TestAxis.Cycle();
gearTestAxis.Cycle();
gearOperation.Cycle();

END_FUNCTION_BLOCK

// ---- Stubs/StubTask.TcPOU
FUNCTION_BLOCK StubTask IMPLEMENTS I_Task
VAR
END_VAR

{warning 'Add method implementation '}
METHOD Abort : BOOL
END_METHOD

{warning 'Add property implementation'}
PROPERTY Busy : BOOL
GET
END_GET
END_PROPERTY

METHOD Cycle : Base_Library.HRESULT
END_METHOD

{warning 'Add property implementation'}
PROPERTY Done : BOOL
GET
END_GET
END_PROPERTY

{warning 'Add property implementation'}
PROPERTY Error : BOOL
GET
END_GET
END_PROPERTY

END_FUNCTION_BLOCK
